FUNCTION F_CreateDynTextDefault : ST_Text
VAR_INPUT
	wsName	: WSTRING;
END_VAR
VAR
END_VAR

F_CreateDynTextDefault.wsNameId := wsName;	
F_CreateDynTextDefault.wsName := wsName;

END_FUNCTION

(* stored: Version 1.1.0.1, ProductVersion 3.1.4024.12
   POU F_CreateDynTextDefault: Id {615e53cb-ab11-4cde-aeb2-762c4aa14925}, SpecialFunc None *)
